SUBAPPLICATION Uebung_004a9 (* mit E_SPLIT_3 *)
  (* Standard: 61499-2; Description: Copyright (c) 2023 Meisterschulen am Ostbahnhof This program and the accompanying materials are made available under the terms of the Eclipse Public License 2.0 which is available at https://www.eclipse.org/legal/epl-2.0/ SPDX-License-Identifier: EPL-2.0 *)
  (* Version 1.0, 2023-10-23, Franz Höpfinger, Meisterschulen am Ostbahnhof *)
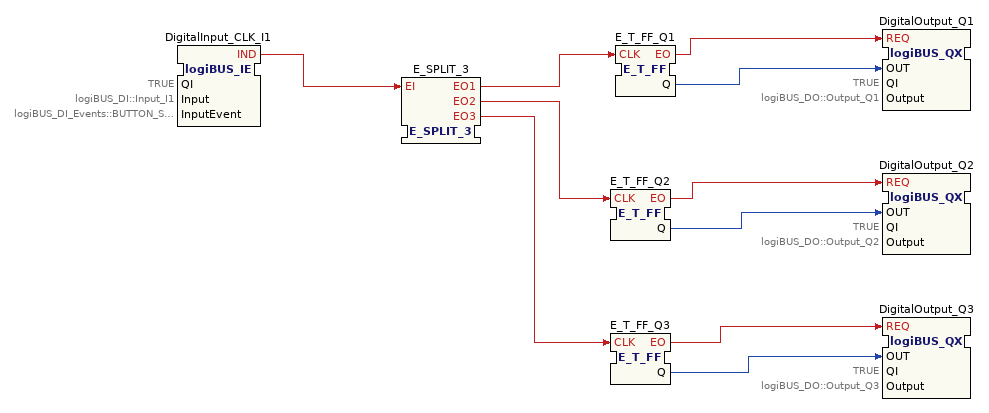
  FBS
    DigitalOutput_Q1 : logiBUS_QX(QI := TRUE, Output := logiBUS_DO::Output_Q1);
    DigitalInput_CLK_I1 : logiBUS_IE(QI := TRUE, Input := logiBUS_DI::Input_I1, InputEvent := logiBUS_DI_Events::BUTTON_SINGLE_CLICK);
    E_T_FF_Q1 : E_T_FF;
    E_T_FF_Q2 : E_T_FF;
    DigitalOutput_Q2 : logiBUS_QX(QI := TRUE, Output := logiBUS_DO::Output_Q2);
    E_SPLIT_3 : E_SPLIT_3;
    E_T_FF_Q3 : E_T_FF;
    DigitalOutput_Q3 : logiBUS_QX(QI := TRUE, Output := logiBUS_DO::Output_Q3);
  END_FBS
  EVENT_CONNECTIONS
    E_T_FF_Q1.EO TO DigitalOutput_Q1.REQ;
    E_T_FF_Q2.EO TO DigitalOutput_Q2.REQ;
    E_SPLIT_3.EO1 TO E_T_FF_Q1.CLK;
    E_SPLIT_3.EO2 TO E_T_FF_Q2.CLK;
    DigitalInput_CLK_I1.IND TO E_SPLIT_3.EI;
    E_T_FF_Q3.EO TO DigitalOutput_Q3.REQ;
    E_SPLIT_3.EO3 TO E_T_FF_Q3.CLK;
  END_CONNECTIONS
  DATA_CONNECTIONS
    E_T_FF_Q1.Q TO DigitalOutput_Q1.OUT;
    E_T_FF_Q2.Q TO DigitalOutput_Q2.OUT;
    E_T_FF_Q3.Q TO DigitalOutput_Q3.OUT;
  END_CONNECTIONS
END_SUBAPPLICATION
